TYPE ST_HexMove_Input :
STRUCT
	t: LREAL;
END_STRUCT
END_TYPE

(* stored: Version 1.1.0.1, ProductVersion 3.1.4020.12
   DUT ST_HexMove_Input: Id {0054867d-7b48-4a4d-9535-53f66c04889b} *)
